{attribute 'reflection'}
FUNCTION_BLOCK FB_LAMP_ONOFF IMPLEMENTS I_LampCtrl
VAR_INPUT
END_VAR
VAR_OUTPUT
END_VAR
VAR
	bOutHw AT%Q*:BOOL;
	
	{attribute 'instance-path'}
	{attribute 'no_init'}
	sPath: STRING;
END_VAR

METHOD OFF : BOOL
// implementation switch Lamp off
OFF := FALSE;

bOutHw := FALSE;
OFF := TRUE;
END_METHOD

METHOD ON : BOOL
// implementation switch Lamp on
ON := FALSE;

bOutHw := TRUE;
ON := TRUE;
END_METHOD

PROPERTY State : string
GET
// additional demo pathname of FB
State := CONCAT('Object: ', sPath); 
State := CONCAT(State, 'State:'); 
State := CONCAT(State, BOOL_TO_STRING(bOutHw));
END_GET
END_PROPERTY

END_FUNCTION_BLOCK

(* stored: Version 1.1.0.1, ProductVersion 3.1.4024.6
   POU FB_LAMP_ONOFF: Id {fc9c48f3-88f3-489b-8472-608355381137}, SpecialFunc None
   Method OFF: Id {b1a6d16c-153d-4d3c-9da5-1782b8fd09df}
   Method ON: Id {152424dd-61ed-47da-a47f-71e6148aa2de}
   Property State: Id {f979ff0a-1114-4932-8462-5a54459d93d7}
   Get Get: Id {22c1d537-2444-47be-a1ac-99d419b7026b} *)
